Staubli VAL3: getPath.pgx

program getPath(string& x_sType[] (dimensions=1))
  local num l_nPos
  local string l_sPath
begin
  // get the TypePath
  l_sPath=x_sType
  do
    l_nPos=find(l_sPath,"/")
    if l_nPos==-1
      l_nPos=find(l_sPath,"\")
    endIf
    if l_nPos!=-1
      l_sPath=right(l_sPath,len(l_sPath)-l_nPos-1)
    endIf
  until l_nPos==-1
  x_sType=l_sPath
end
